PROGRAM MAIN
VAR
END_VAR

END_PROGRAM

(* stored: Version 1.1.0.1, ProductVersion 3.1.4024.12
   POU MAIN: Id {fbdefcff-22c6-41a5-a6dd-64f63b0ba9a4}, SpecialFunc None *)
